// SIMATIC S7-200 SMART project (STEP 7-Micro/WIN SMART), CPU ST30

ORGANIZATION_BLOCK MAIN:OB1
TITLE= 
BEGIN
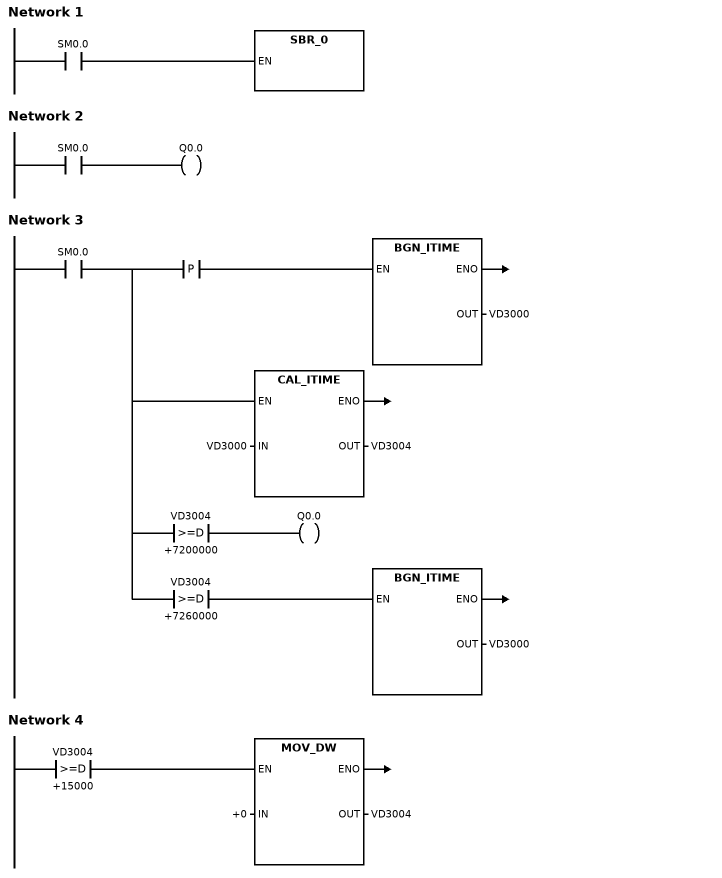
Network 1
// 
// 
LD     SM0.0
CALL   SBR_0:SBR0
Network 2
LD     SM0.0
=      Q0.0
Network 3
LD     SM0.0
LPS
EU
BITIM  VD3000
LRD
CITIM  VD3000, VD3004
LRD
AD>=   VD3004, +7200000
=      Q0.0
LPP
AD>=   VD3004, +7260000
BITIM  VD3000
Network 4
LDD>=  VD3004, +15000
MOVD   +0, VD3004
END_ORGANIZATION_BLOCK

SUBROUTINE_BLOCK SBR_0:SBR0
TITLE= 
// SUBROUTINE COMMENTS
// Press F1 for help and example program
//  
BEGIN
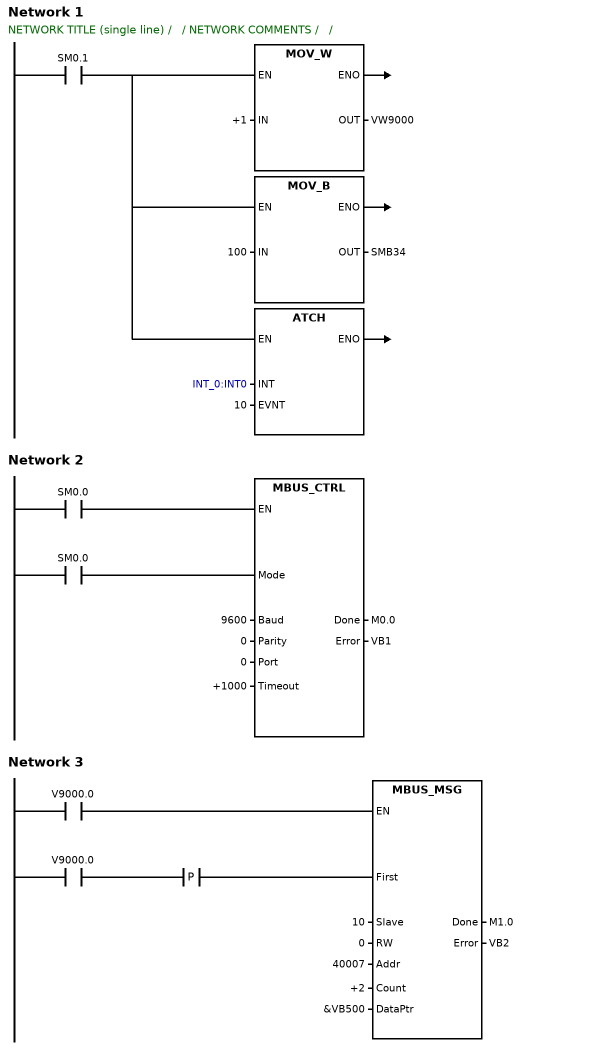
Network 1
// NETWORK TITLE (single line)
//  
// NETWORK COMMENTS
//  
// 
LD     SM0.1
MOVW   +1, VW9000
MOVB   100, SMB34
ATCH   INT_0:INT0, 10
Network 2
LD     SM0.0
=      L60.0
LD     SM0.0
=      L63.7
LD     L60.0
CALL   MBUS_CTRL:SBR1, L63.7, 9600, 0, 0, +1000, M0.0, VB1
Network 3
LD     V9000.0
=      L60.0
LD     V9000.0
EU
=      L63.7
LD     L60.0
CALL   MBUS_MSG:SBR2, L63.7, 10, 0, 40007, +2, &VB500, M1.0, VB2
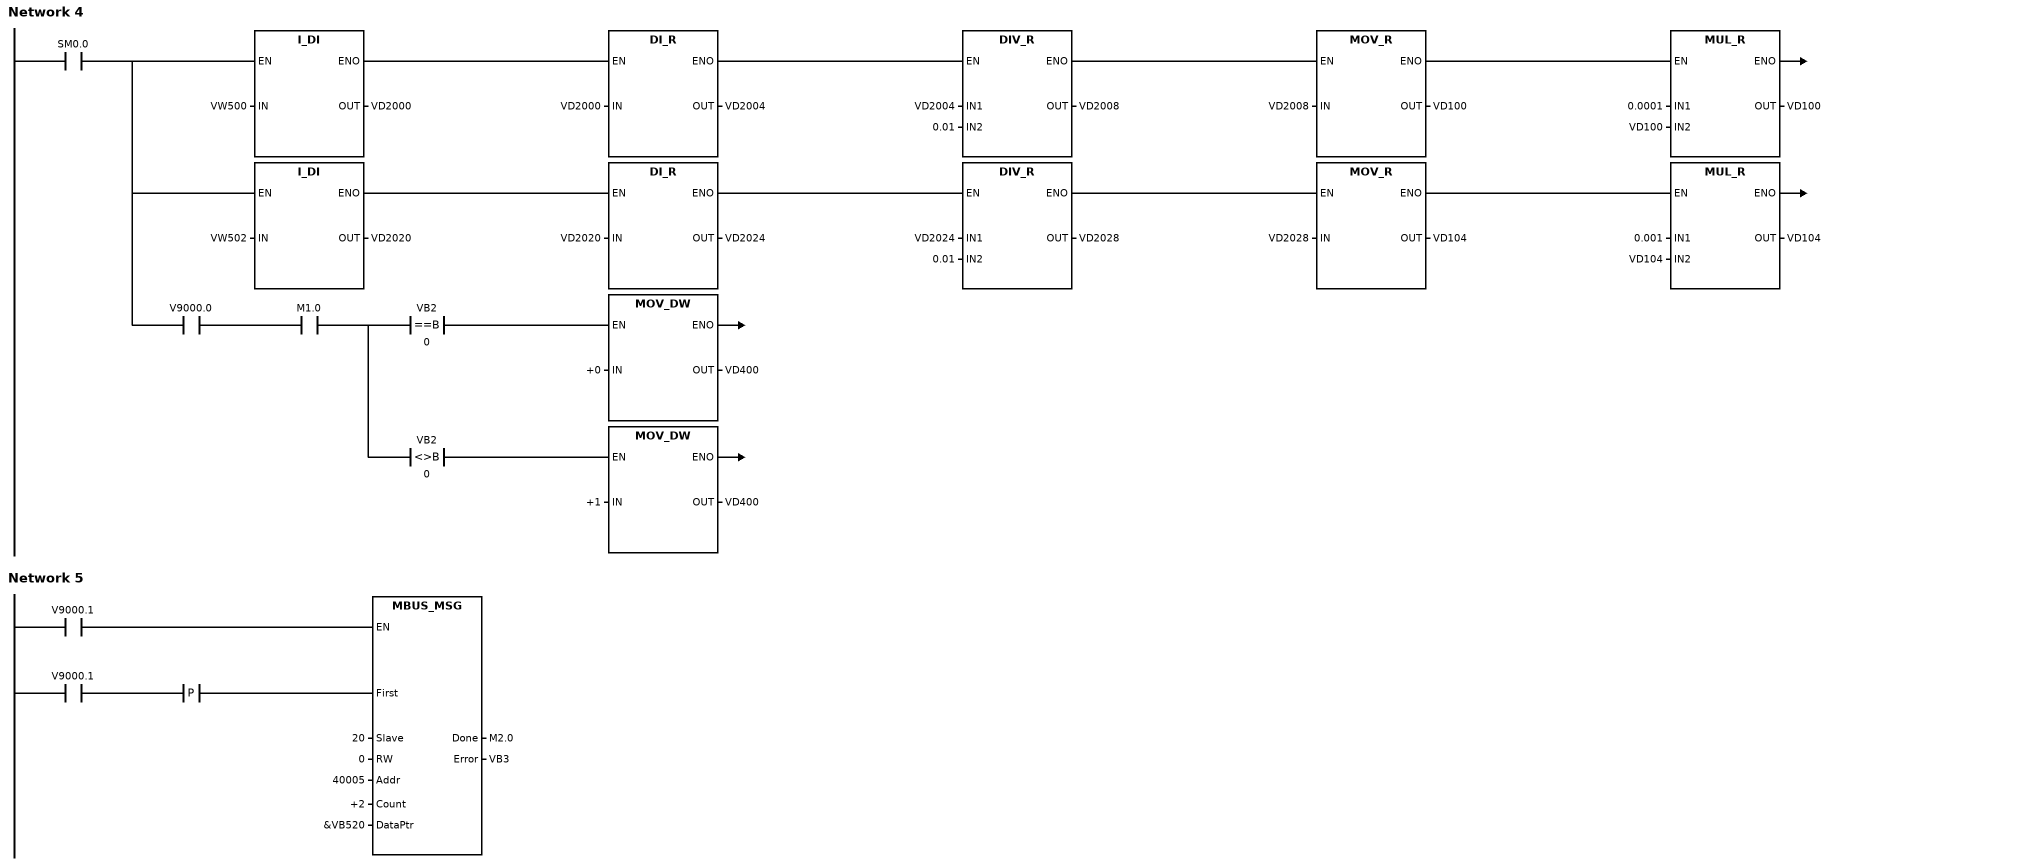
Network 4
LD     SM0.0
LPS
ITD    VW500, VD2000
AENO
DTR    VD2000, VD2004
AENO
MOVR   VD2004, VD2008
AENO
/R     0.01, VD2008
AENO
MOVR   VD2008, VD100
AENO
*R     0.0001, VD100
LRD
ITD    VW502, VD2020
AENO
DTR    VD2020, VD2024
AENO
MOVR   VD2024, VD2028
AENO
/R     0.01, VD2028
AENO
MOVR   VD2028, VD104
AENO
*R     0.001, VD104
LPP
A      V9000.0
A      M1.0
LPS
AB=    VB2, 0
MOVD   +0, VD400
LPP
AB<>   VB2, 0
MOVD   +1, VD400
Network 5
LD     V9000.1
=      L60.0
LD     V9000.1
EU
=      L63.7
LD     L60.0
CALL   MBUS_MSG:SBR2, L63.7, 20, 0, 40005, +2, &VB520, M2.0, VB3
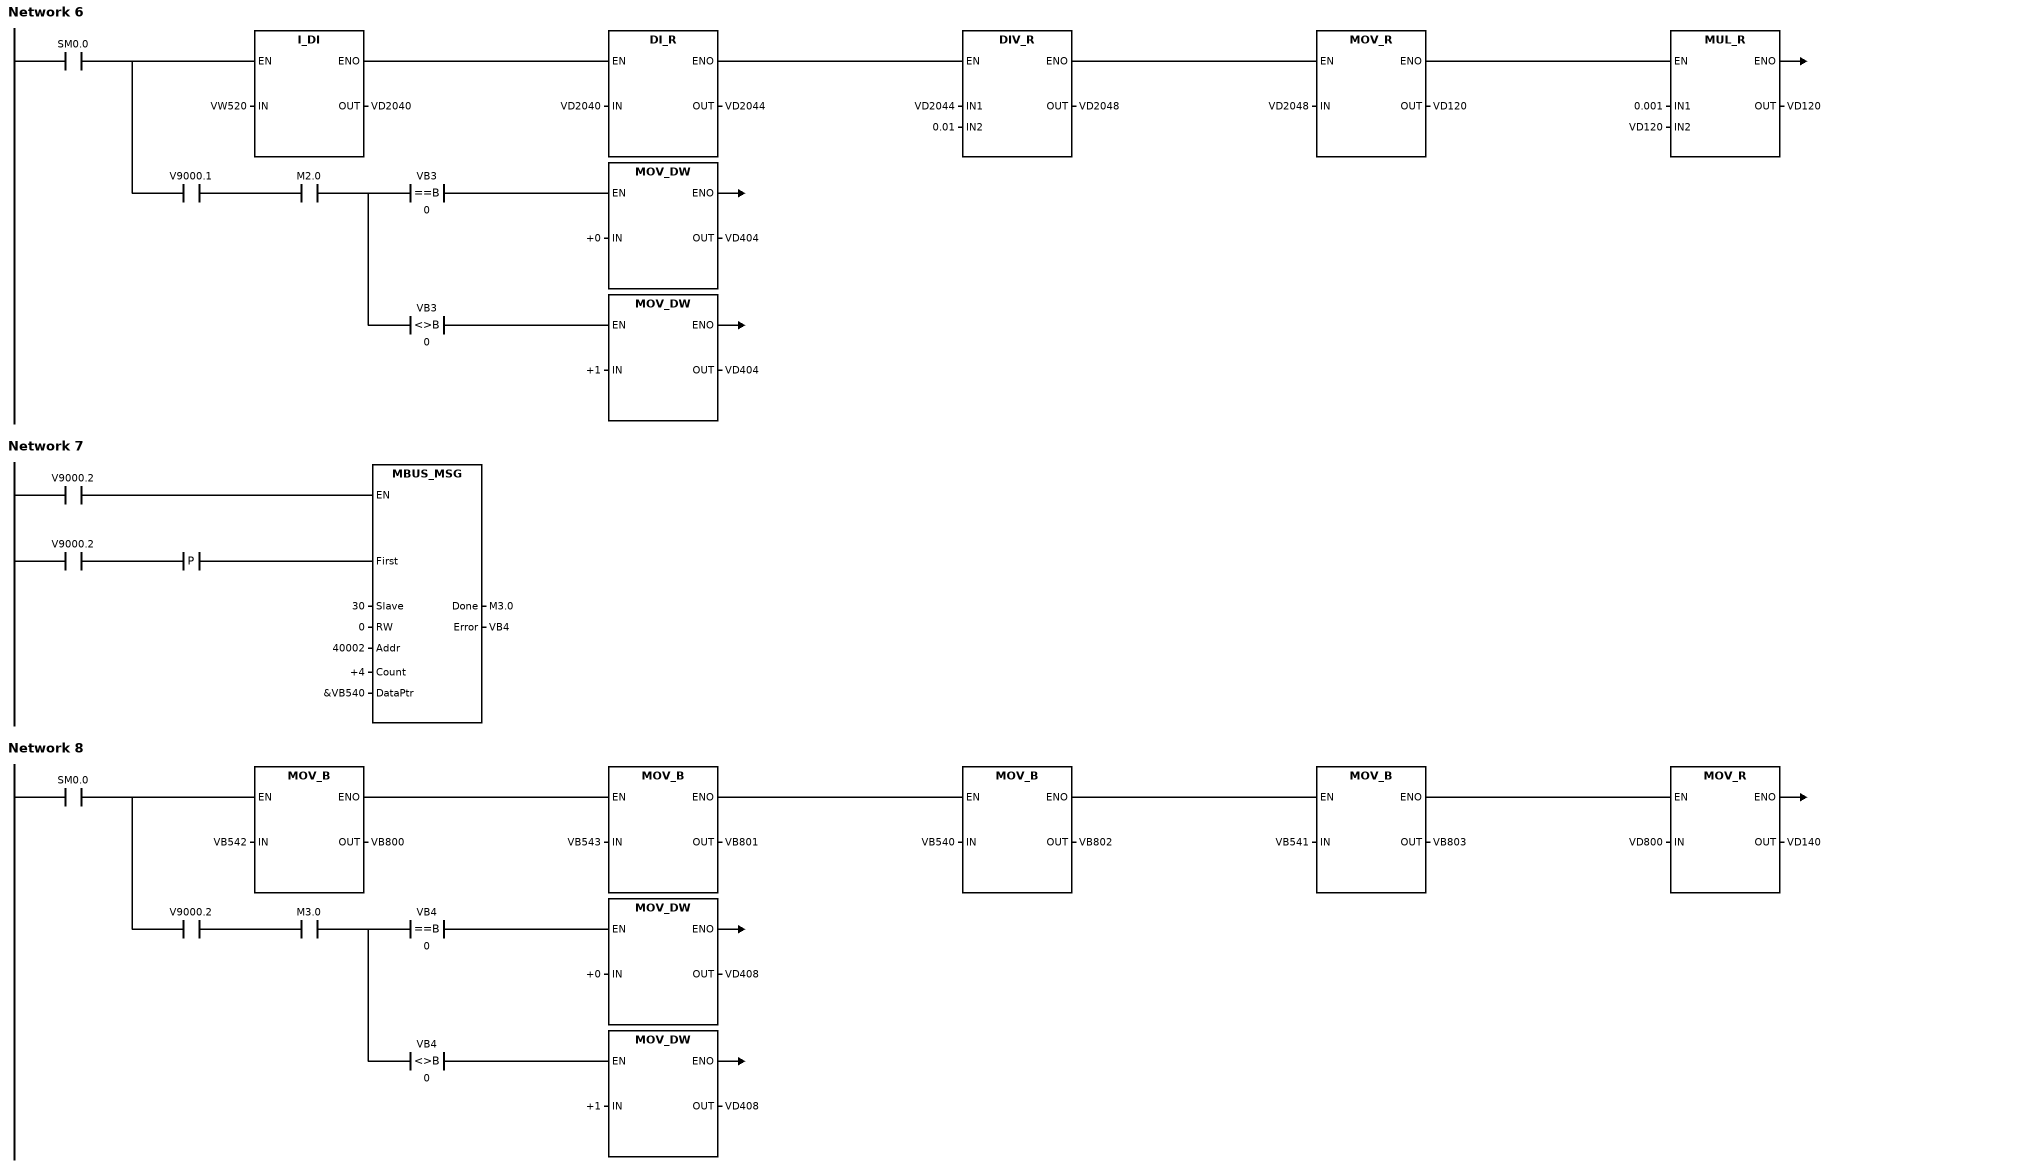
Network 6
LD     SM0.0
LPS
ITD    VW520, VD2040
AENO
DTR    VD2040, VD2044
AENO
MOVR   VD2044, VD2048
AENO
/R     0.01, VD2048
AENO
MOVR   VD2048, VD120
AENO
*R     0.001, VD120
LPP
A      V9000.1
A      M2.0
LPS
AB=    VB3, 0
MOVD   +0, VD404
LPP
AB<>   VB3, 0
MOVD   +1, VD404
Network 7
LD     V9000.2
=      L60.0
LD     V9000.2
EU
=      L63.7
LD     L60.0
CALL   MBUS_MSG:SBR2, L63.7, 30, 0, 40002, +4, &VB540, M3.0, VB4
Network 8
LD     SM0.0
LPS
MOVB   VB542, VB800
AENO
MOVB   VB543, VB801
AENO
MOVB   VB540, VB802
AENO
MOVB   VB541, VB803
AENO
MOVR   VD800, VD140
LPP
A      V9000.2
A      M3.0
LPS
AB=    VB4, 0
MOVD   +0, VD408
LPP
AB<>   VB4, 0
MOVD   +1, VD408
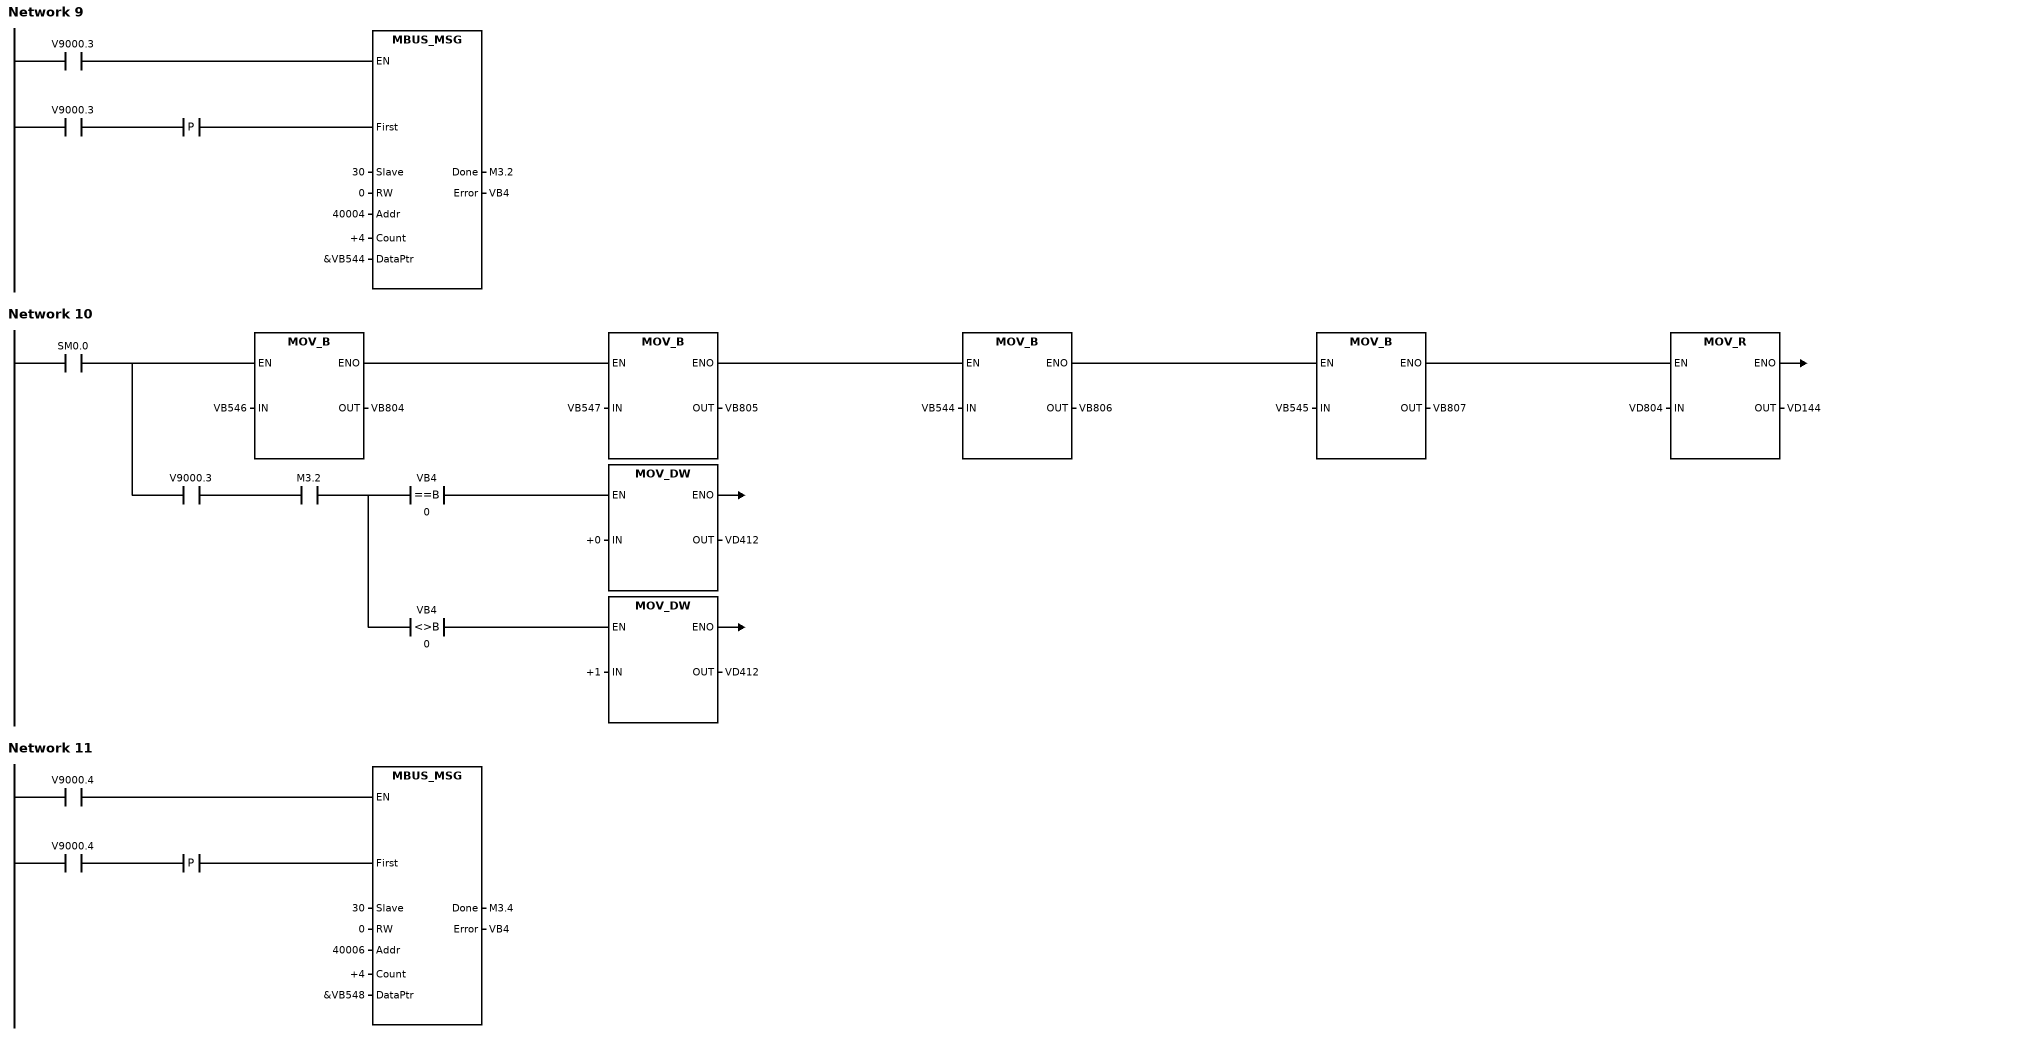
Network 9
LD     V9000.3
=      L60.0
LD     V9000.3
EU
=      L63.7
LD     L60.0
CALL   MBUS_MSG:SBR2, L63.7, 30, 0, 40004, +4, &VB544, M3.2, VB4
Network 10
LD     SM0.0
LPS
MOVB   VB546, VB804
AENO
MOVB   VB547, VB805
AENO
MOVB   VB544, VB806
AENO
MOVB   VB545, VB807
AENO
MOVR   VD804, VD144
LPP
A      V9000.3
A      M3.2
LPS
AB=    VB4, 0
MOVD   +0, VD412
LPP
AB<>   VB4, 0
MOVD   +1, VD412
Network 11
LD     V9000.4
=      L60.0
LD     V9000.4
EU
=      L63.7
LD     L60.0
CALL   MBUS_MSG:SBR2, L63.7, 30, 0, 40006, +4, &VB548, M3.4, VB4
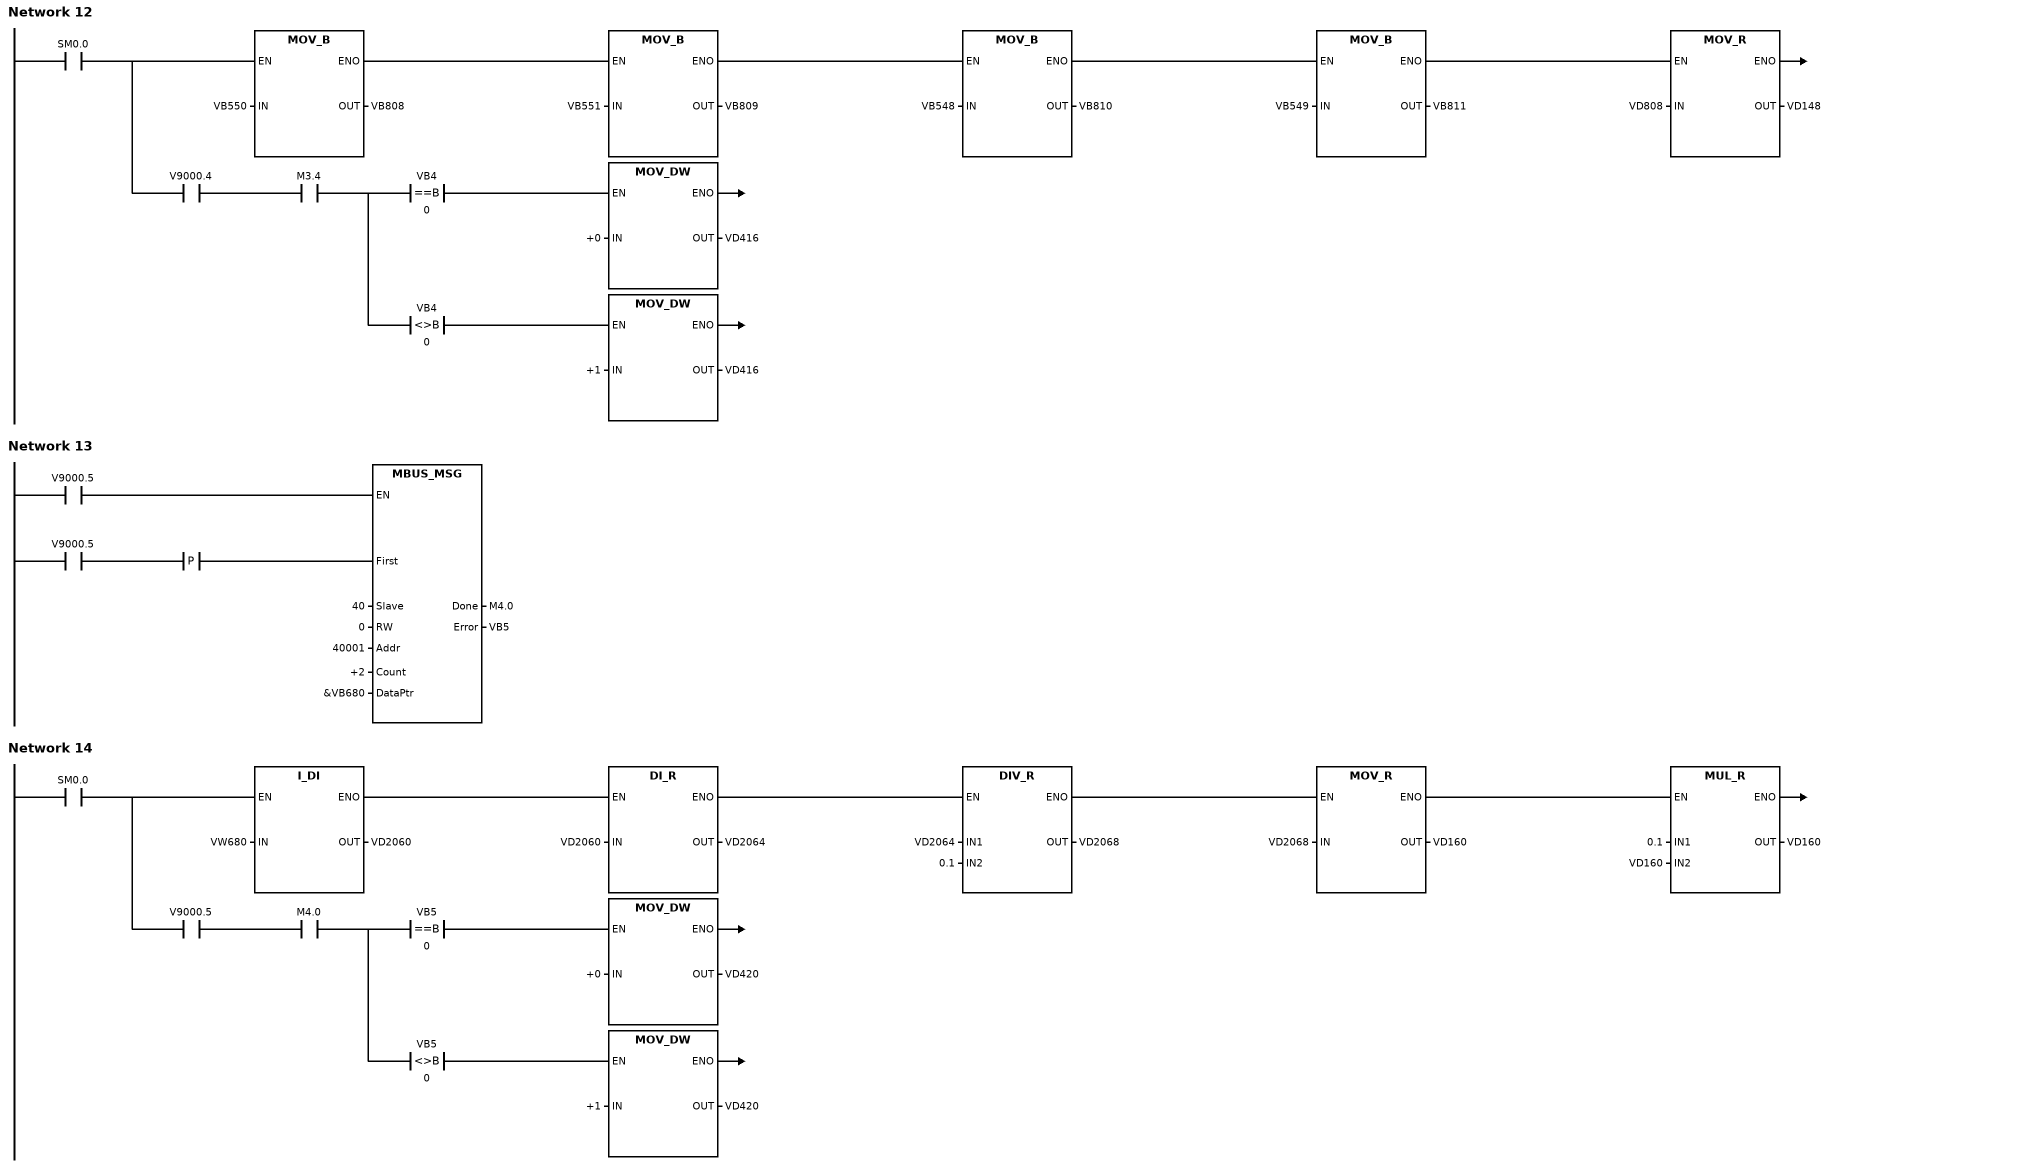
Network 12
LD     SM0.0
LPS
MOVB   VB550, VB808
AENO
MOVB   VB551, VB809
AENO
MOVB   VB548, VB810
AENO
MOVB   VB549, VB811
AENO
MOVR   VD808, VD148
LPP
A      V9000.4
A      M3.4
LPS
AB=    VB4, 0
MOVD   +0, VD416
LPP
AB<>   VB4, 0
MOVD   +1, VD416
Network 13
LD     V9000.5
=      L60.0
LD     V9000.5
EU
=      L63.7
LD     L60.0
CALL   MBUS_MSG:SBR2, L63.7, 40, 0, 40001, +2, &VB680, M4.0, VB5
Network 14
LD     SM0.0
LPS
ITD    VW680, VD2060
AENO
DTR    VD2060, VD2064
AENO
MOVR   VD2064, VD2068
AENO
/R     0.1, VD2068
AENO
MOVR   VD2068, VD160
AENO
*R     0.1, VD160
LPP
A      V9000.5
A      M4.0
LPS
AB=    VB5, 0
MOVD   +0, VD420
LPP
AB<>   VB5, 0
MOVD   +1, VD420
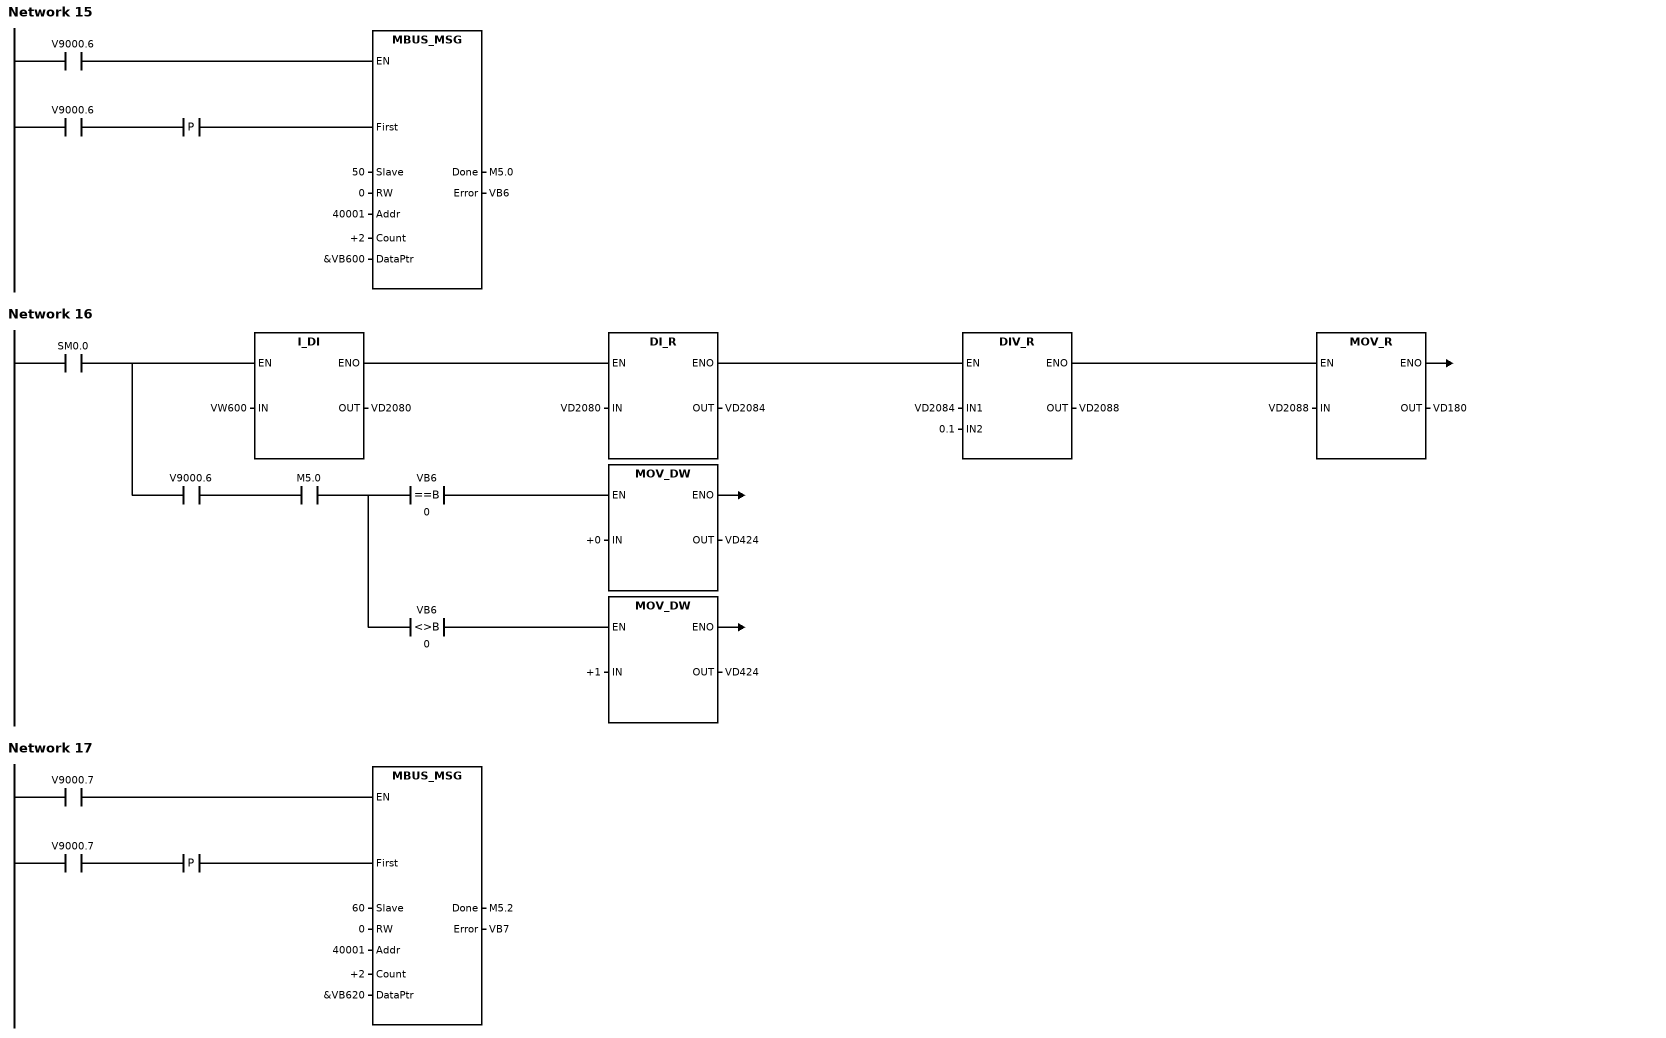
Network 15
LD     V9000.6
=      L60.0
LD     V9000.6
EU
=      L63.7
LD     L60.0
CALL   MBUS_MSG:SBR2, L63.7, 50, 0, 40001, +2, &VB600, M5.0, VB6
Network 16
LD     SM0.0
LPS
ITD    VW600, VD2080
AENO
DTR    VD2080, VD2084
AENO
MOVR   VD2084, VD2088
AENO
/R     0.1, VD2088
AENO
MOVR   VD2088, VD180
LPP
A      V9000.6
A      M5.0
LPS
AB=    VB6, 0
MOVD   +0, VD424
LPP
AB<>   VB6, 0
MOVD   +1, VD424
Network 17
LD     V9000.7
=      L60.0
LD     V9000.7
EU
=      L63.7
LD     L60.0
CALL   MBUS_MSG:SBR2, L63.7, 60, 0, 40001, +2, &VB620, M5.2, VB7
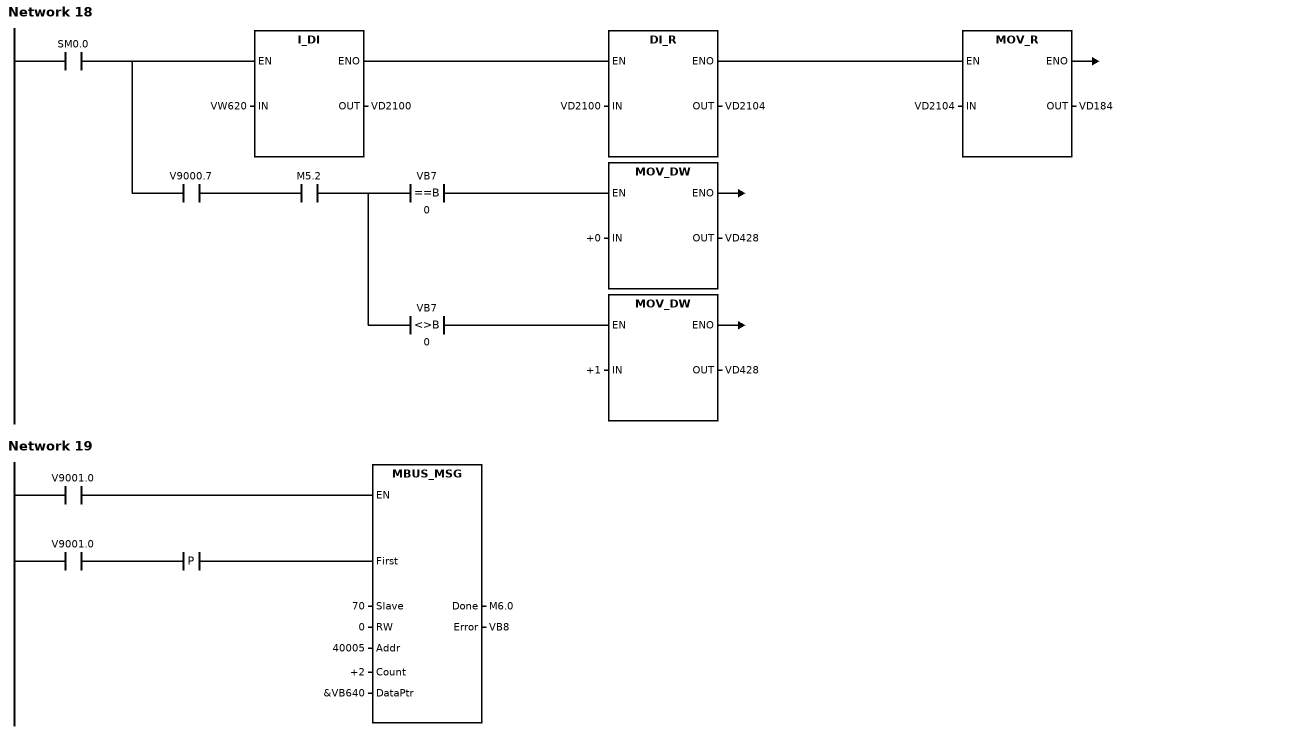
Network 18
LD     SM0.0
LPS
ITD    VW620, VD2100
AENO
DTR    VD2100, VD2104
AENO
MOVR   VD2104, VD184
LPP
A      V9000.7
A      M5.2
LPS
AB=    VB7, 0
MOVD   +0, VD428
LPP
AB<>   VB7, 0
MOVD   +1, VD428
Network 19
LD     V9001.0
=      L60.0
LD     V9001.0
EU
=      L63.7
LD     L60.0
CALL   MBUS_MSG:SBR2, L63.7, 70, 0, 40005, +2, &VB640, M6.0, VB8
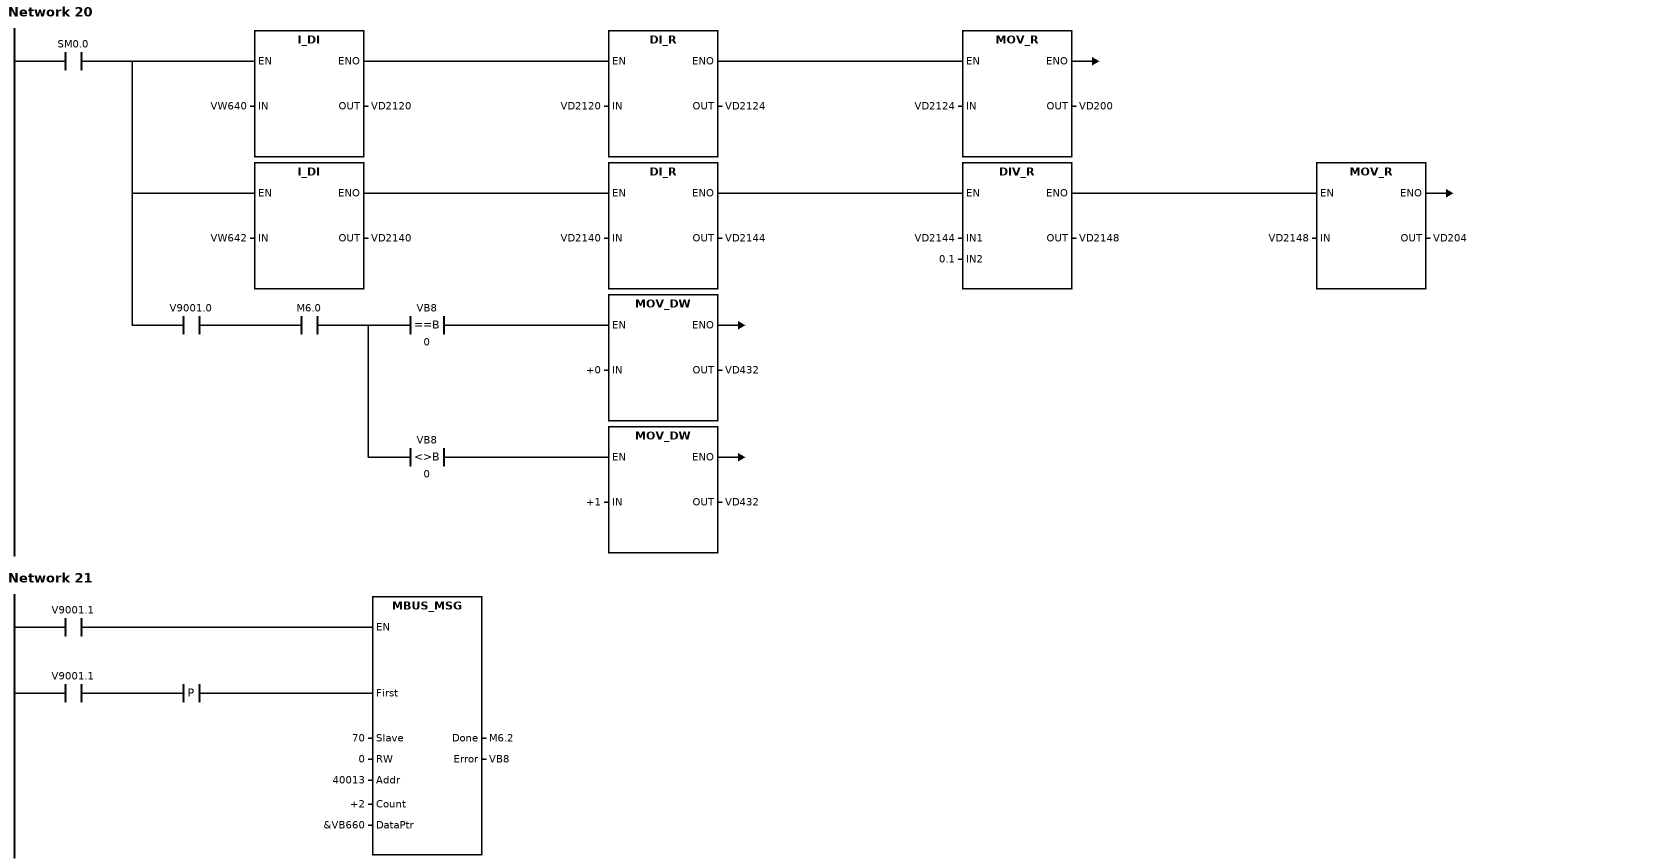
Network 20
LD     SM0.0
LPS
ITD    VW640, VD2120
AENO
DTR    VD2120, VD2124
AENO
MOVR   VD2124, VD200
LRD
ITD    VW642, VD2140
AENO
DTR    VD2140, VD2144
AENO
MOVR   VD2144, VD2148
AENO
/R     0.1, VD2148
AENO
MOVR   VD2148, VD204
LPP
A      V9001.0
A      M6.0
LPS
AB=    VB8, 0
MOVD   +0, VD432
LPP
AB<>   VB8, 0
MOVD   +1, VD432
Network 21
// (network saved uncompiled; LAD cells follow)
// row 0: c0 -| |- V9001.1  c1 --  c2 --  c3 [MBUS_MSG EN:=power@row0, First:=power@row1, Slave:=70, RW:=0, Addr:=40013, Count:=+2, DataPtr:=&VB660, Done=>M6.2, Error=>VB8]
// row 1: c0 -| |- V9001.1  c1 -|P|-  c2 --  c3 [box]
// row 2: c3 [box]
// row 3: c3 [box]
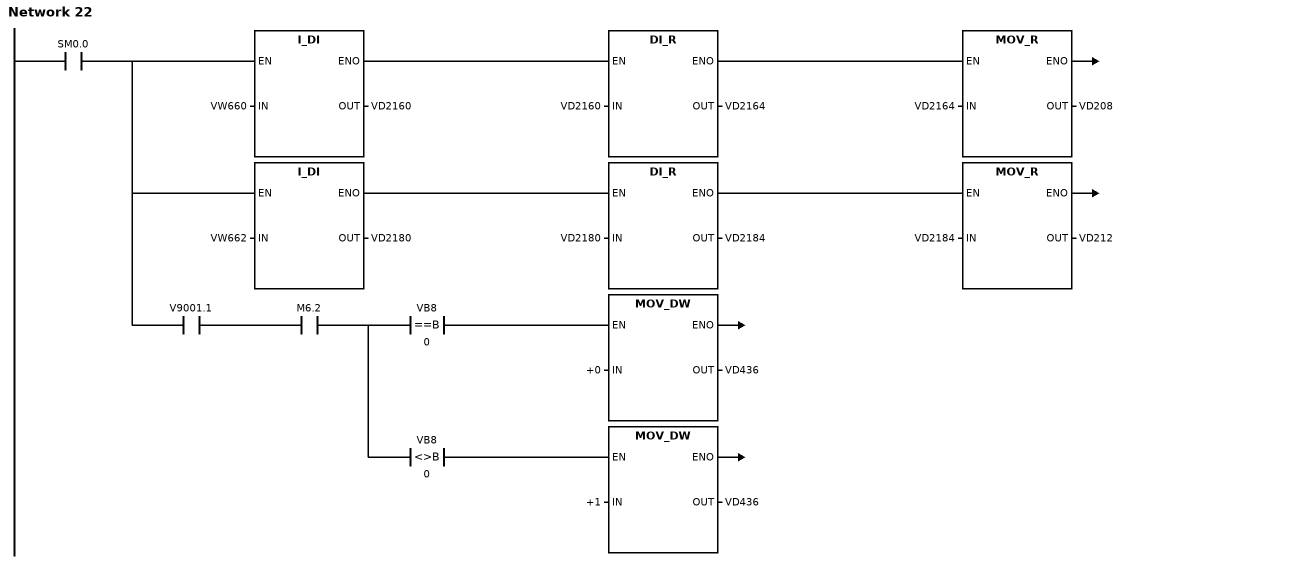
Network 22
LD     SM0.0
LPS
ITD    VW660, VD2160
AENO
DTR    VD2160, VD2164
AENO
MOVR   VD2164, VD208
LRD
ITD    VW662, VD2180
AENO
DTR    VD2180, VD2184
AENO
MOVR   VD2184, VD212
LPP
A      V9001.1
A      M6.2
LPS
AB=    VB8, 0
MOVD   +0, VD436
LPP
AB<>   VB8, 0
MOVD   +1, VD436
END_SUBROUTINE_BLOCK

// SBR1: protected block, not included

// SBR2: protected block, not included

// SBR3: protected block, not included

INTERRUPT_BLOCK INT_0:INT0
TITLE= 
// INTERRUPT ROUTINE COMMENTS
// Press F1 for help and example program
//  
BEGIN
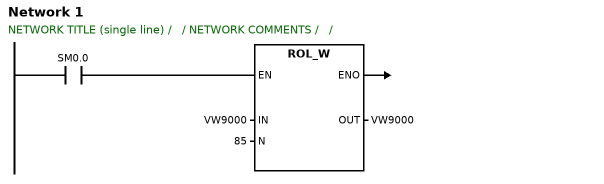
Network 1
// NETWORK TITLE (single line)
//  
// NETWORK COMMENTS
//  
// 
LD     SM0.0
RLW    VW9000, 85
END_INTERRUPT_BLOCK

// INT1: protected block, not included
